// TIA Portal project "2022.06.15_开放式通信2" (V17)

(* hardware
DEVICE "S7-1200 station_1"  S7-1200 Station
   slot 0: "Rack_0"  S7-1200 Rack  Rack  V1.0
   slot 1: "PLC_1"  CPU 1212C DC/DC/DC  6ES7 212-1AE40-0XB0  V4.3
DEVICE "ET 200SP station_1"  ET 200SP-Station
   slot 0: "机架_0"  Rack  6ES5 710-8MAx1
   slot 0: "IO device_1"  IM 155-6 PN ST  6ES7 155-6AU01-0BN0  V4.2
   slot 1: "AQ 2xI ST_1"  AQ 2xI ST  6ES7 135-6GB00-0BA1  V1.0
      slot 1: "AQ 2xI ST_1"  AQ 2xI ST
   slot 2: "AI 2xI 2-,4-wire ST_1"  AI 2xI 2-,4-wire ST  6ES7 134-6GB00-0BA1  V1.0
      slot 1: "AI 2xI 2-,4-wire ST_1"  AI 2xI 2-,4-wire ST
   slot 3: "DQ 8x24VDC/0.5A BA_1"  DQ 8x24VDC/0.5A BA  6ES7 132-6BF00-0AA0  V1.0
      slot 1: "DQ 8x24VDC/0.5A BA_1"  DQ 8x24VDC/0.5A BA
   slot 4: "DI 8x24VDC ST_1"  DI 8x24VDC ST  6ES7 131-6BF01-0BA0  V0.0
      slot 1: "DI 8x24VDC ST_1"  DI 8x24VDC ST
   slot 5: "服务器模块_1"  Server module  6ES7 193-6PA00-0AA0  V1.1
      slot 1: "服务器模块_1"  Server module
   slot 127: "BA 2xRJ45"  BA 2xRJ45  6ES7 193-6AR00-0AA0  V0.0
      slot 1: "Port_1"  X1 P1 R  6ES7 193-6AR00-0AA0  V0.0
      slot 2: "Port_2"  X1 P2 R  6ES7 193-6AR00-0AA0  V0.0
*)

// ===== PLC "PLC_1"  CPU 1212C DC/DC/DC =====

VAR_GLOBAL   // PLC tag table "默认变量表"
   "Tag_1" AT %I2.0 : Bool;
   "Tag_2" AT %Q2.0 : Bool;
   "Tag_3" AT %IW68 : Word;
   "Tag_4" AT %QW64 : Word;
END_VAR

ORGANIZATION_BLOCK "Main"   // OB1, LAD, ProgramCycle
TITLE = "Main Program Sweep (Cycle)"
{ S7_Optimized_Access := 'TRUE' }
VERSION : 0.1
   VAR_INPUT
      Initial_Call : Bool;   // Initial call of this OB
      Remanence : Bool;   // =True, if remanent data are available
   END_VAR
BEGIN

REGION Network 1
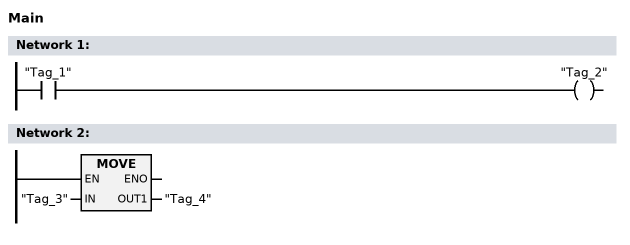
   RUNG wire#powerrail
      Contact( "Tag_1" )
      Coil( "Tag_2" )
   END_RUNG
   // the same network as SCL:
   "Tag_2" := "Tag_1";
END_REGION

REGION Network 2
   RUNG wire#powerrail
      Move(in := "Tag_3", out1 => "Tag_4")
   END_RUNG
   // the same network as SCL:
   "Tag_4" := "Tag_3";
END_REGION
END_ORGANIZATION_BLOCK